FUNCTION_BLOCK PAEActMixingValve EXTENDS PAEActuator2way_Analog
VAR_INPUT
END_VAR
VAR_OUTPUT
END_VAR
VAR
END_VAR

METHOD PUBLIC PAEActMixingValve
VAR_INPUT
END_VAR
END_METHOD

END_FUNCTION_BLOCK

(* stored: Version 1.1.0.1, ProductVersion 3.1.4020.12
   POU PAEActMixingValve: Id {fd1cd2b8-5582-4c3f-8213-b0d131d14be4}, SpecialFunc None
   Method PAEActMixingValve: Id {4607e9a4-e8f4-42e1-bd0c-e29111fcb1f1} *)
